{attribute 'qualified_only'}
VAR_GLOBAL CONSTANT
	MAX_ILOSC_ELEMENTOW						: INT := 10; //Ilementów głównych
	MAX_ILOSC_ZDARZEN_NA_ELEMENT			: INT := 10;
	MAX_ILOSC_ELEMENTOW_NA_PODZESPOL		: INT := 10;
	MAX_ILOSC_ZDARZEN						: INT := 100;
	MAX_ILOSC_ZDARZEN_DO_WYSWIETLANIA		: INT := 50;
END_VAR

(* stored: Version 1.1.0.1, ProductVersion 3.1.4024.11
   GVL GVL_LogowanieBledow_Stale: Id {6f7cf282-1cc0-47c3-a879-cb2e9534c558} *)
